INTERFACE ITF_Observable

METHOD notifyObserverConnection : BOOL
END_METHOD

METHOD registerObserver : BOOL
VAR_INPUT
	Observer : ITF_Observer;
END_VAR
END_METHOD

METHOD removeObserver : BOOL
VAR_INPUT
	Observer : ITF_Observer;
END_VAR
END_METHOD

END_INTERFACE

(* stored: Version 1.1.0.1, ProductVersion 3.1.4024.12
   Itf ITF_Observable: Id {299ee042-88c5-4516-be13-3cb87c805b06}
   Method notifyObserverConnection: Id {7d400b0a-b618-4ff9-ac85-a4b5079a0b8f}
   Method registerObserver: Id {245a0123-2057-4f43-b962-4dd2985459f0}
   Method removeObserver: Id {dc591c9c-1963-4568-ad86-73c64d0c48b1} *)
